FUNCTION_BLOCK FB_OPCUA_ReadOrWriteNode IMPLEMENTS I_OPCUA_WorkOnNode
VAR_INPUT
END_VAR
VAR_OUTPUT
	busy: BOOL;
	error : BOOL;
END_VAR
VAR

	fbUA_Read			: UA_Read;
	stNodeAddInfo			: ST_UANodeAdditionalInfo;
	cbData_R				: UDINT;
	
	iState		: INT;
	nErrorID	: DWORD;
	dataAdd : PVOID;
	lastErrorStep: INT;
	readToggle : FB_ToggleHeartBeat;
	Executing : BOOL;
	writeStep : INT;
	(* Declarations for UA_Write *)
	fbUA_Write : UA_Write; 
	
	(* Declarations for UA_NodeReleaseHandle *)
	fbUA_NodeReleaseHandle : UA_NodeReleaseHandle;
	
	(* Other declarations *) 
	errorID : DWORD;	
	clientVariablePrev : BYTE;
	firstTimeWrite : BOOL;
		fbUA_NodeGetHandle : UA_NodeGetHandle;
	NodeID : ST_UANodeID;
	nNodeHdl : DWORD;
END_VAR

{warning 'add method implementation '}
METHOD read : BOOL
VAR_INPUT
	{attribute 'anytypeclass' := 'ANY'}
	clientVariable	: ANY;
	(* VAR_INFO of the target variable (from GVL_OPC)*)
	clientVariableInfo	: __SYSTEM.VAR_INFO;
	serverNodeIdentifier	: STRING;
	nameSpaceLocationIdentifierEx	: STRING(MAX_STRING_LENGTH);
	ConnectionHdl	: DWORD;
	nNamespaceIndex			: UINT;
END_VAR
CASE istate OF
0: (* Compile node id's *)
//	FOR node := 1 TO 4 DO
//		IF clientVariable[node] <> '' THEN
//			NodeIds[node].eIdentifierType := eUAIdentifierType_String;
//			NodeIDs[node].nNamespaceIndex := nNamespaceIndex;
//			NodeIDs[node].sIdentifier	:= CONCAT(nameSpaceLocationIdentifierEx ,clientVariable[node]);
//		END_IF
//		IF node = 4 THEN
			error := FALSE;
			nNodeHdl :=0;
			Executing := TRUE;
			iState := iState + 1;
//		END_IF
//	END_FOR

	
1:	(* Get Node Handle *)
	
		(* UA_NodeGetHandle *)
		NodeID.eIdentifierType := eUAIdentifierType_String;
		NodeID.nNamespaceIndex := nNamespaceIndex;
		NodeID.sIdentifier := CONCAT(nameSpaceLocationIdentifierEx,serverNodeIdentifier);
		fbUA_NodeGetHandle(
		  Execute := TRUE,
		  ConnectionHdl := connectionHdl,
		  NodeID := NodeID,
		  NodeHdl => nNodeHdl);
		IF NOT fbUA_NodeGetHandle.Busy THEN
		  fbUA_NodeGetHandle(Execute := FALSE);
		  IF NOT fbUA_NodeGetHandle.Error THEN
			istate := istate + 1;
		  ELSE
			//Executing := FALSE;
			//error := TRUE;
			errorID := fbUA_NodeGetHandle.ErrorID;
			istate := 3;
		  END_IF
		END_IF

	
2: 	(* UA_Read *)

	dataAdd := ADR(clientVariable);
	fbUA_Read(
		  Execute := TRUE,
		  ConnectionHdl := connectionHdl,
		  NodeHdl := nNodeHdl,
		  cbData := SIZEOF(clientVariable),//clientVariableInfo.BitSize,
		stNodeAddInfo 	:= stNodeAddInfo,
		  pVariable :=clientVariableInfo.ByteAddress	
		);

	IF NOT fbUA_Read.Busy THEN
//		readToggle(I_TimeIntervalSecs := 0.1);
//		IF readTOggle.O_Update THEN
			fbUA_Read( Execute := FALSE, cbData_R => cbData_R);
//		END_IF
		//fbUA_ReadList( Execute := FALSE, cbData_R => cbData_R);

		IF NOT fbUA_Read.Error THEN
			(* session closed *)
			//iState 		:= iState + 1; 
			iState 		:= 3;
		ELSE
			//bError		:= TRUE;
			//error := TRUE;
			lastErrorStep := 2;
			nErrorID	:= fbUA_Read.ErrorID;
			iState 		:= 3; (* idle *)
		END_IF
	END_IF


3:	(* Release Node Handle *)
		fbUA_NodeReleaseHandle(
			Execute			:= TRUE,
			ConnectionHdl	:= ConnectionHdl,
			NodeHdl			:= nNodeHdl
		);
	
		IF NOT fbUA_NodeReleaseHandle.Busy THEN
			fbUA_NodeReleaseHandle(Execute := FALSE);
	
			IF NOT fbUA_NodeReleaseHandle.Error THEN
				Executing := FALSE;
				istate := 0;
			ELSE
				//Executing := FALSE;
				//error		:= TRUE;
				error := TRUE;
				errorID	:= fbUA_NodeReleaseHandle.ErrorID;
				istate 	:= 0; (* idle *)
			END_IF
		END_IF
END_CASE
busy := Executing;
END_METHOD

{warning 'add method implementation '}
METHOD write : BOOL
VAR_INPUT
	{attribute 'anytypeclass' := 'ANY'}
	clientVariable	: ANY;
	(* VAR_INFO of the target variable (from GVL_OPC)*)
	clientVariableInfo	: __SYSTEM.VAR_INFO;
	serverNodeIdentifier	: STRING;
	nameSpaceLocationIdentifierEx	: STRING(MAX_STRING_LENGTH);
	connectionHdl: DWORD;
	nNamespaceIndex			: UINT;
END_VAR
CASE writeStep OF
	
	0:
		error := FALSE;
		IF clientVariable.pValue^ <> clientVariablePrev OR NOT firstTimeWrite THEN
//		IF clientVariable.pValue <> clientVariablePrev OR NOT firstTimeWrite THEN
			Executing := TRUE;
			clientVariablePrev := clientVariable.pValue^;
			writeStep := 1;
		END_IF
	
	  1: 
//		Executing := TRUE;
		(* UA_NodeGetHandle *)
		NodeID.eIdentifierType := eUAIdentifierType_String;
		NodeID.nNamespaceIndex := nNamespaceIndex;
		NodeID.sIdentifier := CONCAT(nameSpaceLocationIdentifierEx,serverNodeIdentifier);
		fbUA_NodeGetHandle(
		  Execute := TRUE,
		  ConnectionHdl := connectionHdl,
		  NodeID := NodeID,
		  NodeHdl => nNodeHdl);
		IF NOT fbUA_NodeGetHandle.Busy THEN
		  fbUA_NodeGetHandle(Execute := FALSE);
		  IF NOT fbUA_NodeGetHandle.Error THEN
			writeStep := writeStep + 1;
		  ELSE
			//Executing := FALSE;
			//error := TRUE;
			errorID := fbUA_NodeGetHandle.ErrorID;
			writeStep := 2;
		  END_IF
		END_IF
	  2: (* UA_Write *)
//		writeDone := FALSE;
		fbUA_Write(
		  Execute := TRUE,
		  ConnectionHdl := connectionHdl,
		  NodeHdl := nNodeHdl,
		  stNodeAddInfo := stNodeAddInfo,
		  cbData := clientVariableInfo.BitSize,
		  pVariable := clientVariableInfo.ByteAddress);
		IF NOT fbUA_Write.Busy THEN
		  fbUA_Write(
			Execute := FALSE,
			pVariable := clientVariableInfo.ByteAddress);
		
		  IF NOT fbUA_Write.Error THEN
//				writeDone := TRUE;
			//writeStep := writeStep + 1;
				writeStep := 3;
		  ELSE
			//Executing := FALSE;
			error := TRUE;
			errorID := fbUA_Write.ErrorID;
			writeStep := 3;
		  END_IF
		END_IF
	3:	(* Release Node Handle *)
		fbUA_NodeReleaseHandle(
			Execute			:= TRUE,
			ConnectionHdl	:= ConnectionHdl,
			NodeHdl			:= nNodeHdl
		);
	
		IF NOT fbUA_NodeReleaseHandle.Busy THEN
			fbUA_NodeReleaseHandle(Execute := FALSE);
	
			IF NOT fbUA_NodeReleaseHandle.Error THEN
				firstTimeWrite := TRUE;
//				clientVariablePrev := clientVariable.pValue^;
				Executing := FALSE;
				writeStep := 0;
			ELSE
				//Executing := FALSE;
				//error		:= TRUE;
				error := TRUE;
				errorID	:= fbUA_NodeReleaseHandle.ErrorID;
				writeStep 	:= 0; (* idle *)
			END_IF
		END_IF
END_CASE
busy := Executing ;
END_METHOD

END_FUNCTION_BLOCK

(* stored: Version 1.1.0.1, ProductVersion 3.1.4024.9
   POU FB_OPCUA_ReadOrWriteNode: Id {0e3c7aeb-71ed-4c55-86bf-e2c7680b355d}, SpecialFunc None
   Method read: Id {03c3b3f3-09be-48e8-a71a-d9f38d3c1c07}
   Method write: Id {64b5c044-7dd9-4728-a1be-b684ca04e6b0} *)
